(* PLC project Unnamed, Unknown Unnamed 1 *)
(* stored: creationDateTime 2026-01-05T14:16:15, modificationDateTime 2026-01-05T14:16:15 *)

PROGRAM main
  VAR_INPUT
    X0 : BOOL;
    X1 : BOOL;
    X2 : BOOL;
    X3 : BOOL;
    X4 : BOOL;
    X5 : BOOL;
  END_VAR
  VAR_OUTPUT
    Y0 : BOOL;
    Y1 : BOOL;
  END_VAR

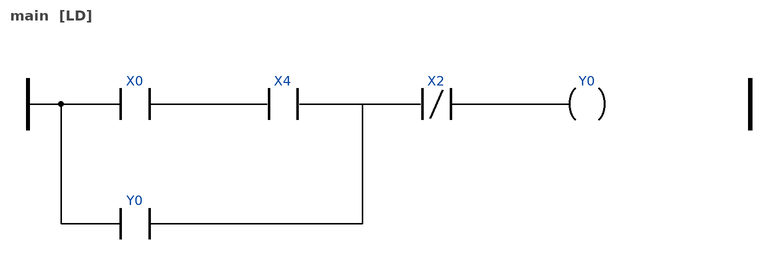
(* LD diagram, written out as Structured Text *)
Y0 := (X0 AND X4 OR Y0) AND NOT X2;
END_PROGRAM

CONFIGURATION Config0
  RESOURCE Res0 ON PLC
    TASK task0(INTERVAL := T#20ms, PRIORITY := 1);
    PROGRAM instance0 WITH task0 : main;
  END_RESOURCE
END_CONFIGURATION
